// TIA Portal V17 export
// export: Created 2023-12-22T15:28:36.5102018Z, ExportSetting WithDefaults, DisplayName Totally Integrated Automation Portal, DisplayVersion V17, DisplayName TIA Portal Openness, DisplayVersion V17, DisplayName TIA Portal Version Control Interface, DisplayVersion V17, DisplayName STEP 7 Professional, DisplayVersion V17, DisplayName STEP 7 Safety, DisplayVersion V17, DisplayName WinCC Advanced, DisplayVersion V17
DATA_BLOCK "PID_example_DB"   // DB900
VERSION : 0.1
// stored: AutoNumber false, DBAccessibleFromOPCUA true, InstanceOfName PID_ex, InstanceOfType FB
"PID_ex"
   // VAR_INPUT
   //    Start : Bool;
   //    SP_A : Real;
   //    Value : Real;
   // END_VAR
   // VAR_OUTPUT
   //    PWM : Bool;
   //    Result : Real;
   // END_VAR
   // VAR RETAIN
   //    CMD { S7_SetPoint := 'True'} : "CMD";
   //    SP_M : Real;
   //    SP : Real;
   //    x { S7_SetPoint := 'True'} : Real;
   //    SP_x : Real;
   //    Value_x : Real;
   //    Buffer : Real;
   //    PID_Output : Real;
   //    PID_Hand : Real;
   //    Sys : Struct
   //       Err_Ack : Bool;
   //       Alm_SP_H : Bool;
   //       Alm_SP_L : Bool;
   //       Alm_In_H : Bool;
   //       Alm_In_L : Bool;
   //       Activate : Bool;
   //       Error_code : DWord;
   //       Warning_code : DWord;
   //       "Type" : Int;
   //       State : Int;
   //       Mode : Int;
   //    END_STRUCT;
   //    Settings : Struct
   //       SP_P { S7_SetPoint := 'True'} : Real;
   //       SP_Ti { S7_SetPoint := 'True'} : Real;
   //       SP_Td { S7_SetPoint := 'True'} : Real;
   //       SP_Cycle { S7_SetPoint := 'True'} : Real;
   //       Max_SP { S7_SetPoint := 'True'} : Real;
   //       Min_SP { S7_SetPoint := 'True'} : Real;
   //       Max_in { S7_SetPoint := 'True'} : Real;
   //       Min_in { S7_SetPoint := 'True'} : Real;
   //       Max_out { S7_SetPoint := 'True'} : Real;
   //       Min_out { S7_SetPoint := 'True'} : Real;
   //       DeadBand { S7_SetPoint := 'True'} : Real;
   //       Max : Real;
   //       Min : Real;
   //    END_STRUCT;
   //    PID { S7_SetPoint := 'True'} : PID_Compact;
   //    Converter : "Converter";
   //    Conveter_Back : "Converter";
   //    C { S7_SetPoint := 'True'} : "Time_R";
   //    pos : Array[0..15] of Bool;
   // END_VAR
BEGIN
END_DATA_BLOCK
